INTERFACE ITF_DigOut

METHOD set : BOOL
VAR_INPUT
	state : BOOL;
END_VAR
END_METHOD

END_INTERFACE

(* stored: Version 1.1.0.1, ProductVersion 3.1.4026.8
   Itf ITF_DigOut: Id {616324e0-884a-4236-a920-f1e73764f81b}
   Method set: Id {42007418-5013-445e-9db0-a9a06da55375} *)
